{attribute 'linkalways'} 
{attribute 'no_explicit_call' := 'This FB is a CLASS and must be accessed using methods or properties'}
{attribute 'enable_dynamic_creation'}
FUNCTION_BLOCK FINAL ASIN_LREAL EXTENDS Node
VAR
	in : _LREAL(0.0);
	out : _LREAL(0.0);
END_VAR

METHOD PUBLIC Clone : I_Node
VAR
	pNode : POINTER TO ASIN_LREAL;
END_VAR
pNode := __NEW(ASIN_LREAL);
Clone := pNode^;
END_METHOD

METHOD FB_init : BOOL
VAR_INPUT
	bInitRetains : BOOL; // if TRUE, the retain variables are initialized (warm start / cold start)
	bInCopyCode : BOOL;  // if TRUE, the instance afterwards gets moved into the copy code (online change)
END_VAR
AddInput('in',THIS^.in);
AddOutput('out', THIS^.out);
END_METHOD

METHOD PROTECTED OnExecute
VAR
END_VAR
out.Value := ASIN(in.Value);
END_METHOD

END_FUNCTION_BLOCK

(* stored: Version 1.1.0.1, ProductVersion 3.1.4024.15
   POU ASIN_LREAL: Id {20db0292-cc32-4483-9713-6ac185faea30}, SpecialFunc None
   Folder Constructor: Id {a24fc4ef-1280-4691-a767-1d29a78e52b9}
   Method Clone: Id {2495b32b-d91a-405b-825b-61374968506b}
   Method FB_init: Id {3a1b808c-33bd-4be7-bcbe-ba4475d983e7}
   Method OnExecute: Id {6ba390ef-0a72-42f5-a7a0-064826115c93} *)
